(* Logix 5000 project; controller Reto2IOT vendor 1 type 14 code 156 rev 30.11; software revision 30.00 *)

TASK MainTask (continuous, watchdog 500 ms) : MainProgram

MODULES
   Local : vendor 1 type 14 code 156 (Compact 0, rev 30.11)
      DIG_IN : 1769-IQ16 (Compact 4, rev 1.1, Input RPI 20 ms)
      ANALOG_OUT : vendor 1 type 10 code 48 (Compact 3, rev 1.1, Output RPI 80 ms)
      DIG_OUT : vendor 1 type 7 code 86 (Compact 5, rev 2.1, Output RPI 20 ms)
      ANALOG_IN : vendor 1 type 10 code 44 (Compact 2, rev 2.1, Output RPI 80 ms)
      DEVICENET : vendor 1 type 12 code 105 (Compact 1, rev 1.1, Output RPI 20 ms)
END_MODULES

VAR_GLOBAL   (* controller tags *)
   BandaCorrecta : BOOL;
   Bandera : BOOL;
   BanderaA : BOOL;
   BanderaV : BOOL;
   BanSenA : BOOL;
   BanSenV : BOOL;
   ContadorA : COUNTER := (PRE := 100);
   ContadorV : COUNTER := (PRE := 100);
   FIO_AvanzarA : BOOL := 1;
   FIO_AvanzarUPA : BOOL := 1;
   FIO_AvanzarUPV : BOOL := 1;
   FIO_AvanzarV : BOOL := 1;
   FIO_DetenerA : BOOL;
   FIO_DetenerV : BOOL;
   FIO_I0 : BOOL;
   FIO_I10 : BOOL := 1;
   FIO_I11 : BOOL := 1;
   FIO_I12 : BOOL;
   FIO_I3 : BOOL;
   FIO_I4 : BOOL;
   FIO_I6 : BOOL;
   FIO_I7 : BOOL;
   FIO_I8 : BOOL;
   FIO_Iniciar : BOOL;
   FIO_km1 : BOOL;
   FIO_O0 : BOOL;
   FIO_O1 : BOOL;
   FIO_O2 : BOOL;
   FIO_O3 : BOOL;
   FIO_O4 : BOOL;
   FIO_O5 : BOOL;
   FIO_ParadaUPA : BOOL;
   FIO_ParadaUPV : BOOL;
   FIO_Start : BOOL;
   FIO_Stop : BOOL;
   FIO_Stop_emergencia : BOOL;
   FlancoBajadaA : BOOL;
   FlancoBajadaV : BOOL;
   GD_INPUT_0 : BOOL;
   GD_INPUT_1 : BOOL;
   GD_INPUT_2 : BOOL;
   GD_OUT_0 : BOOL;
   GD_OUT_1 : BOOL;
   Km1 : ALIAS FOR Local:5:O.Data.0;
   Prueba : BOOL;
   PusherA : ALIAS FOR Local:5:O.Data.2;
   PusherV : ALIAS FOR Local:5:O.Data.3;
   Start : ALIAS FOR Local:4:I.Data.1;
   Stop : ALIAS FOR Local:4:I.Data.0;
   Timer_TA : TIMER := (PRE := 5000, ACC := 5000);
   Timer_TV : TIMER := (PRE := 5000, ACC := 5000);
   TimerAvan : TIMER := (PRE := 1000, EN := 1, TT := 1);
   TimerAvanV : TIMER := (PRE := 1000, EN := 1, TT := 1);
   TimerBien : TIMER := (PRE := 500);
   TimerExitA : TIMER := (PRE := 1000, ACC := 1000);
   TimerExitV : TIMER := (PRE := 1000, ACC := 1000);
   TimerInicio : TIMER := (PRE := 2000, ACC := 2000, EN := 1, DN := 1);
   TimerInicioV : TIMER := (PRE := 2000, ACC := 2000, EN := 1, DN := 1);
   TimerP : TIMER := (PRE := 4000);
   TimerPUN : TIMER := (PRE := 3000, ACC := 2000, TT := 1, DN := 1);
   TimerPUNV : TIMER := (PRE := 3000, ACC := 2000, TT := 1, DN := 1);
   TimerPV : TIMER := (PRE := 4000);
END_VAR

PROGRAM MainProgram   (* main routine MainRoutine *)

ROUTINE Azul   (* ladder *)
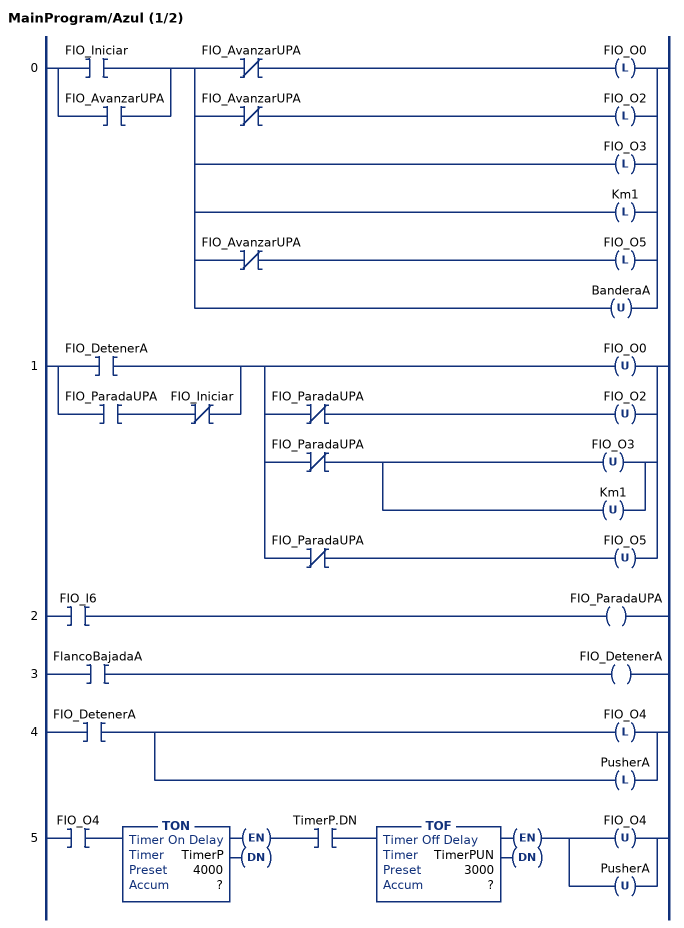
   0: [XIC(FIO_Iniciar) ,XIC(FIO_AvanzarUPA) ][XIO(FIO_AvanzarUPA) OTL(FIO_O0) ,XIO(FIO_AvanzarUPA) OTL(FIO_O2) ,[OTL(FIO_O3) ,OTL(Km1) ] ,XIO(FIO_AvanzarUPA) OTL(FIO_O5) ,OTU(BanderaA) ];
   1: [XIC(FIO_DetenerA) ,XIC(FIO_ParadaUPA) XIO(FIO_Iniciar) ][OTU(FIO_O0) ,XIO(FIO_ParadaUPA) OTU(FIO_O2) ,XIO(FIO_ParadaUPA) [OTU(FIO_O3) ,OTU(Km1) ] ,XIO(FIO_ParadaUPA) OTU(FIO_O5) ];
   2: XIC(FIO_I6)OTE(FIO_ParadaUPA);
   3: XIC(FlancoBajadaA)OTE(FIO_DetenerA);
   4: XIC(FIO_DetenerA)[OTL(FIO_O4) ,OTL(PusherA) ];
   5: XIC(FIO_O4)TON(TimerP,?,?)XIC(TimerP.DN)TOF(TimerPUN,?,?)[OTU(FIO_O4) ,OTU(PusherA) ];
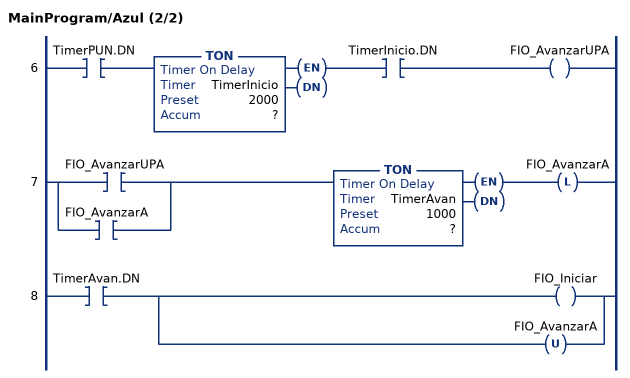
   6: XIC(TimerPUN.DN)TON(TimerInicio,?,?)XIC(TimerInicio.DN)OTE(FIO_AvanzarUPA);
   7: [XIC(FIO_AvanzarUPA) ,XIC(FIO_AvanzarA) ]TON(TimerAvan,?,?)OTL(FIO_AvanzarA);
   8: XIC(TimerAvan.DN)[OTE(FIO_Iniciar) ,OTU(FIO_AvanzarA) ];
END_ROUTINE

ROUTINE MainRoutine   (* ladder *)
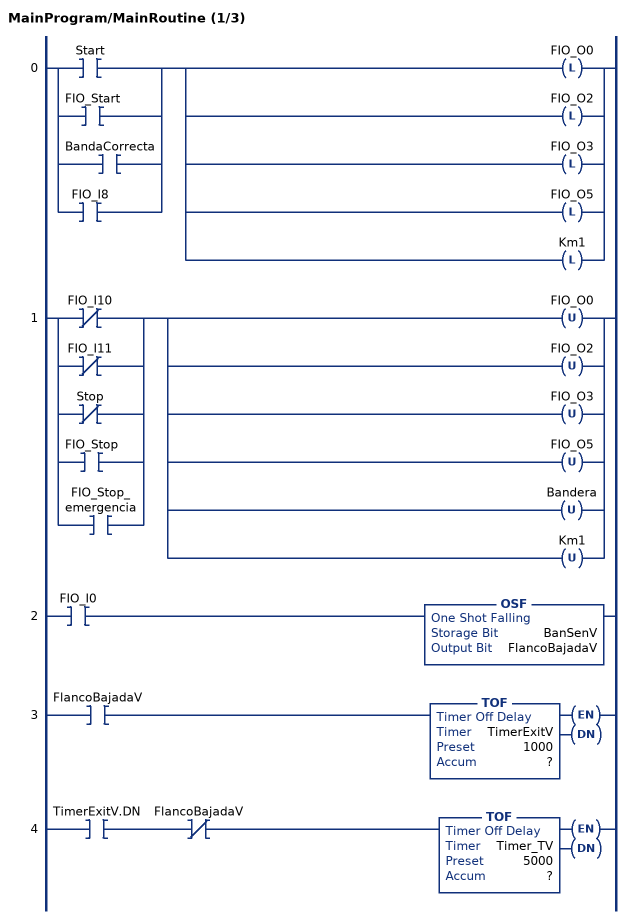
   0: [XIC(Start) ,XIC(FIO_Start) ,XIC(BandaCorrecta) ,XIC(FIO_I8) ][OTL(FIO_O0) ,OTL(FIO_O2) ,OTL(FIO_O3) ,OTL(FIO_O5) ,OTL(Km1) ];
   1: [XIO(FIO_I10) ,XIO(FIO_I11) ,XIO(Stop) ,XIC(FIO_Stop) ,XIC(FIO_Stop_emergencia) ][OTU(FIO_O0) ,OTU(FIO_O2) ,OTU(FIO_O3) ,OTU(FIO_O5) ,OTU(Bandera) ,OTU(Km1) ];
   2: XIC(FIO_I0)OSF(BanSenV,FlancoBajadaV);
   3: XIC(FlancoBajadaV)TOF(TimerExitV,?,?);
   4: XIC(TimerExitV.DN)XIO(FlancoBajadaV)TOF(Timer_TV,?,?);
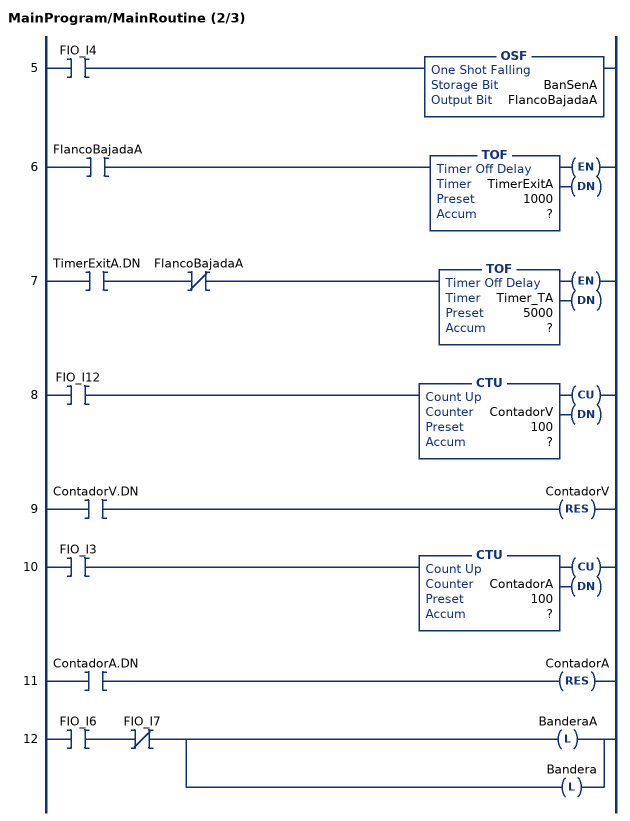
   5: XIC(FIO_I4)OSF(BanSenA,FlancoBajadaA);
   6: XIC(FlancoBajadaA)TOF(TimerExitA,?,?);
   7: XIC(TimerExitA.DN)XIO(FlancoBajadaA)TOF(Timer_TA,?,?);
   8: XIC(FIO_I12)CTU(ContadorV,?,?);
   9: XIC(ContadorV.DN)RES(ContadorV);
   10: XIC(FIO_I3)CTU(ContadorA,?,?);
   11: XIC(ContadorA.DN)RES(ContadorA);
   12: XIC(FIO_I6)XIO(FIO_I7)[OTL(BanderaA) ,OTL(Bandera) ];
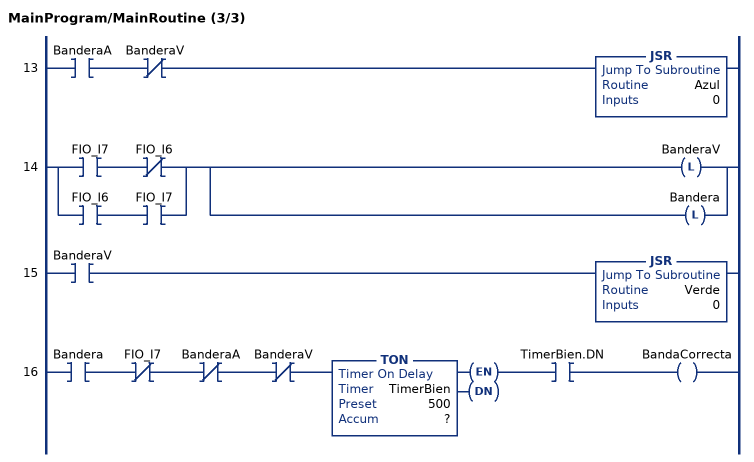
   13: XIC(BanderaA)XIO(BanderaV)JSR(Azul,0);
   14: [XIC(FIO_I7) XIO(FIO_I6) ,XIC(FIO_I6) XIC(FIO_I7) ][OTL(BanderaV) ,OTL(Bandera) ];
   15: XIC(BanderaV)JSR(Verde,0);
   16: XIC(Bandera)XIO(FIO_I7)XIO(BanderaA)XIO(BanderaV)TON(TimerBien,?,?)XIC(TimerBien.DN)OTE(BandaCorrecta);
END_ROUTINE

ROUTINE Verde   (* ladder *)
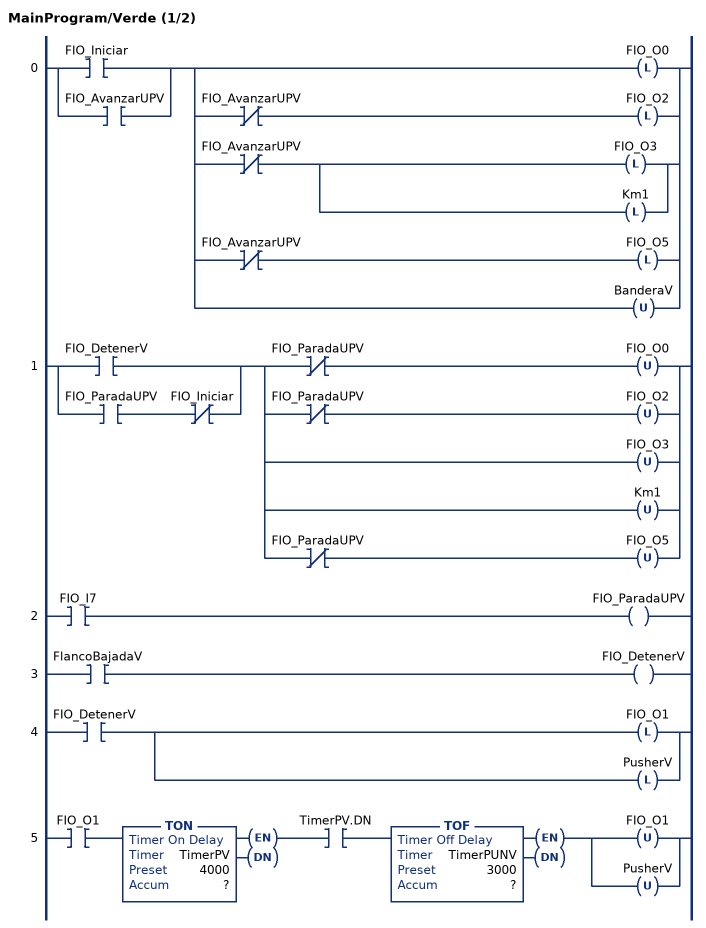
   0: [XIC(FIO_Iniciar) ,XIC(FIO_AvanzarUPV) ][OTL(FIO_O0) ,XIO(FIO_AvanzarUPV) OTL(FIO_O2) ,XIO(FIO_AvanzarUPV) [OTL(FIO_O3) ,OTL(Km1) ] ,XIO(FIO_AvanzarUPV) OTL(FIO_O5) ,OTU(BanderaV) ];
   1: [XIC(FIO_DetenerV) ,XIC(FIO_ParadaUPV) XIO(FIO_Iniciar) ][XIO(FIO_ParadaUPV) OTU(FIO_O0) ,XIO(FIO_ParadaUPV) OTU(FIO_O2) ,[OTU(FIO_O3) ,OTU(Km1) ] ,XIO(FIO_ParadaUPV) OTU(FIO_O5) ];
   2: XIC(FIO_I7)OTE(FIO_ParadaUPV);
   3: XIC(FlancoBajadaV)OTE(FIO_DetenerV);
   4: XIC(FIO_DetenerV)[OTL(FIO_O1) ,OTL(PusherV) ];
   5: XIC(FIO_O1)TON(TimerPV,?,?)XIC(TimerPV.DN)TOF(TimerPUNV,?,?)[OTU(FIO_O1) ,OTU(PusherV) ];
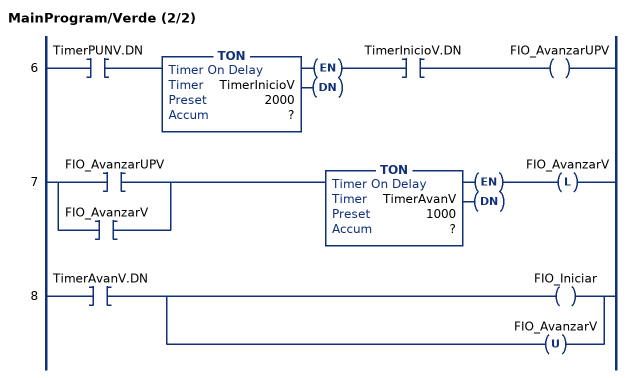
   6: XIC(TimerPUNV.DN)TON(TimerInicioV,?,?)XIC(TimerInicioV.DN)OTE(FIO_AvanzarUPV);
   7: [XIC(FIO_AvanzarUPV) ,XIC(FIO_AvanzarV) ]TON(TimerAvanV,?,?)OTL(FIO_AvanzarV);
   8: XIC(TimerAvanV.DN)[OTE(FIO_Iniciar) ,OTU(FIO_AvanzarV) ];
END_ROUTINE
END_PROGRAM
